TYPE EL3154_PDOS :
	STRUCT
		
		HwToPLC : EL3154_HWTOPLC_PDOS;
		
	END_STRUCT
END_TYPE

(* stored: Version 1.1.0.1, ProductVersion 3.1.4024.15
   DUT EL3154_PDOS: Id {514fb89d-5250-44a3-99fd-6c503144cda8} *)
